# EPICS autosave request: stdApp/Db/scaler_channelN_settings.req
# FILE... Jscaler_channelN_settings.req
# USAGE.. Jscaler.db fields autosave'd.
$(P)$(S).NM$(Ch)
$(P)$(S).PR$(Ch)
$(P)$(S).G$(Ch)
